TYPE DUT_STRUCT_C000004_PROD :
STRUCT
	sCellName			:STRING := 'C000004';
	sIpAddress			:STRING := '10.38.190.201';
	sAmsNetId			:STRING := '10.38.190.201.1.1';
	sOpcUaURL			:STRING := 'opc.tcp://10.38.190.201:4840';
	sStation1			:STRING := 'S000003';
END_STRUCT
END_TYPE

(* stored: Version 1.1.0.1, ProductVersion 3.1.4024.5
   DUT DUT_STRUCT_C000004_PROD: Id {43d8e211-6c80-43c0-be2f-7bd22946e0fc} *)
